FUNCTION_BLOCK FB_LightTowerComponent IMPLEMENTS I_LightTowerComponent
VAR_INPUT
	component : REFERENCE TO BOOL;
END_VAR
VAR
	_component	: ZigaLibs_Core.BoolEx := (variable := component);
END_VAR

_component(variable := component);

METHOD Activate
IF NOT __ISVALIDREF(component) THEN
	RETURN;
END_IF
_component.Set();
END_METHOD

METHOD Deactivate
IF NOT __ISVALIDREF(component) THEN
	RETURN;
END_IF
_component.Reset();
END_METHOD

METHOD FB_init : BOOL
VAR_INPUT
	bInitRetains : BOOL; // if TRUE, the retain variables are initialized (warm start / cold start)
	bInCopyCode : BOOL;  // if TRUE, the instance afterwards gets moved into the copy code (online change)
END_VAR
END_METHOD

METHOD PulseWithInterval
VAR_INPUT
	DurationOn	: TIME;
	DurationOff	: TIME;
END_VAR
VAR_INST
	timerOn		: Tc2_Standard.TON;
	timerOff	: Tc2_Standard.TON;
END_VAR
IF NOT __ISVALIDREF(component) THEN
	RETURN;
END_IF
_component.PulseWithInterval(DurationOn,DurationOff);
END_METHOD

{attribute 'monitoring':='call'}
(* Gets the current state of the component*)
PROPERTY Value : BOOL
GET
Value := _component.Value;
END_GET
END_PROPERTY

END_FUNCTION_BLOCK

(* stored: Version 1.1.0.1, ProductVersion 3.1.4024.14
   POU FB_LightTowerComponent: Id {7b461e9f-dfac-0508-356d-25a618b18337}, SpecialFunc None
   Method Activate: Id {5642512f-163a-04c4-3e94-b83af68483c6}
   Method Deactivate: Id {c1bb4cd8-3ce5-01d0-1d8f-99f05e888c8c}
   Method FB_init: Id {5d69ceb3-5a24-071f-2087-acc3b0b0fc39}
   Method PulseWithInterval: Id {f2a2e1f2-763f-0c67-28c6-1c86551f52f9}
   Property Value: Id {8552b7bb-5e13-0828-24b4-1980ad6d5e83}
   Get Get: Id {ae9e4849-b1e7-0d41-2158-59ecdab7c37d} *)
